// TIA Portal project "CPU1500_Profinet_PLC1_PLC2" (V16)

(* hardware
DEVICE "Station S71500/ET200MP_1"  S7-1500 station
   slot 0: "Châssis_0"  Rack  6ES7 590-1***0-0AA0
   slot 1: "PLC_1"  CPU 1511-1 PN  6ES7 511-1AK02-0AB0  V2.5
      slot 3: "Ecran CPU_1"  6ES7591-1AA00-0AA0
      slot 32768: "Interface PROFINET_1"  X1
         slot 32769: "Port_1"  X1 P1
         slot 32770: "Port_2"  X1 P2
   slot 2: "DI 32x24VDC BA_1"  DI 32x24VDC BA  6ES7 521-1BL10-0AA0  V1.0
   slot 3: "DQ 32x24VDC/0.5A BA_1"  DQ 32x24VDC/0.5A BA  6ES7 522-1BL10-0AA0  V1.0
DEVICE "Station S71500/ET200MP_2"  S7-1500 station
   slot 0: "Châssis_0"  Rack  6ES7 590-1***0-0AA0
   slot 1: "PLC_2"  CPU 1511-1 PN  6ES7 511-1AK01-0AB0  V2.1
      slot 3: "Ecran CPU_1"  6ES7591-1AA00-0AA0
      slot 32768: "Interface PROFINET_1"  X1
         slot 32769: "Port_1"  X1 P1
         slot 32770: "Port_2"  X1 P2
*)

// ===== PLC "PLC_1"  CPU 1511-1 PN =====

VAR_GLOBAL   // PLC tag table "Table de variables standard"
   "Clock_Byte" AT %MB0 : Byte;
   "Clock_10Hz" AT %M0.0 : Bool;
   "Clock_5Hz" AT %M0.1 : Bool;
   "Clock_2.5Hz" AT %M0.2 : Bool;
   "Clock_2Hz" AT %M0.3 : Bool;
   "Clock_1.25Hz" AT %M0.4 : Bool;
   "Clock_1Hz" AT %M0.5 : Bool;
   "Clock_0.625Hz" AT %M0.6 : Bool;
   "Clock_0.5Hz" AT %M0.7 : Bool;
END_VAR

DATA_BLOCK "DB_EMISSION"   // DB1
{ S7_Optimized_Access := 'FALSE' }
VERSION : 0.1
   VAR
      BOOL_0 : Bool;
      BOOL_1 : Bool;
      BOOL_2 : Bool;
      BOOL_3 : Bool;
      BOOL_4 : Bool;
      BOOL_5 : Bool;
      BOOL_6 : Bool;
      BOOL_7 : Bool;
      INT_0 : Int;
      INT_1 : Int;
      INT_2 : Int;
      INT_3 : Int;
      DINT_0 : DInt;
      DINT_1 : DInt;
      DINT_2 : DInt;
      DINT_3 : DInt;
   END_VAR
BEGIN
END_DATA_BLOCK

DATA_BLOCK "DB_RECEPTION"   // DB2
{ S7_Optimized_Access := 'FALSE' }
VERSION : 0.1
   VAR
      BOOL_0 : Bool;
      BOOL_1 : Bool;
      BOOL_2 : Bool;
      BOOL_3 : Bool;
      BOOL_4 : Bool;
      BOOL_5 : Bool;
      BOOL_6 : Bool;
      BOOL_7 : Bool;
      BOOL_8 : Bool;
      BOOL_9 : Bool;
      BOOL_10 : Bool;
      BOOL_11 : Bool;
      BOOL_12 : Bool;
      BOOL_13 : Bool;
      BOOL_14 : Bool;
      BOOL_15 : Bool;
      INT_0 : Int;
      INT_1 : Int;
      INT_2 : Int;
      INT_3 : Int;
      INT_4 : Int;
      INT_5 : Int;
      DINT_0 : DInt;
      DINT_1 : DInt;
      DINT_2 : DInt;
      DINT_3 : DInt;
      DINT_4 : DInt;
      DINT_5 : DInt;
      DINT_6 : DInt;
      DINT_7 : DInt;
      DINT_8 : DInt;
      DINT_9 : DInt;
      DINT_10 : DInt;
      DINT_11 : DInt;
   END_VAR
BEGIN
END_DATA_BLOCK

FUNCTION "FC_GEST_COM" : Void   // FC1, LAD
{ S7_Optimized_Access := 'TRUE' }
VERSION : 0.1
BEGIN

REGION Network 1
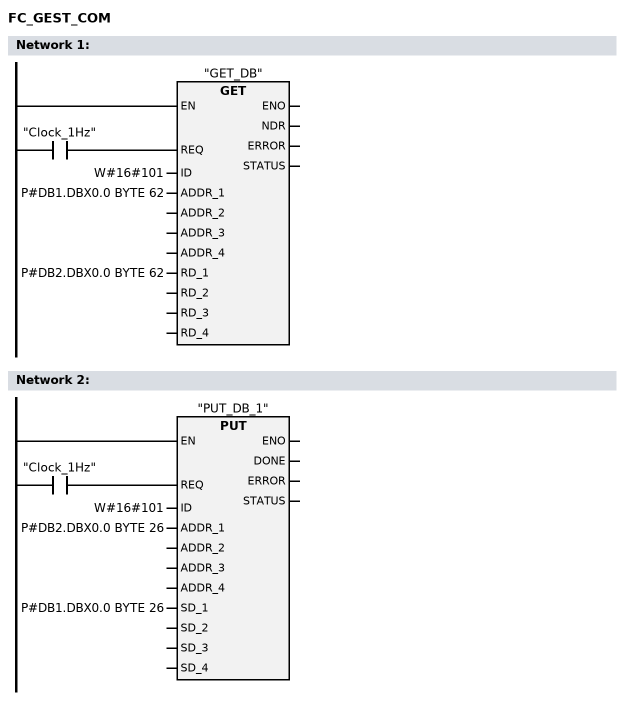
   "GET_DB"(REQ := "Clock_1Hz", ID := W#16#101, ADDR_1 := P#DB1.DBX0.0 BYTE 62, RD_1 := P#DB2.DBX0.0 BYTE 62);   // GET
END_REGION

REGION Network 2
   "PUT_DB_1"(REQ := "Clock_1Hz", ID := W#16#101, ADDR_1 := P#DB2.DBX0.0 BYTE 26, SD_1 := P#DB1.DBX0.0 BYTE 26);   // PUT
END_REGION
END_FUNCTION

ORGANIZATION_BLOCK "Main"   // OB1, LAD, ProgramCycle
TITLE = "Main Program Sweep (Cycle)"
{ S7_Optimized_Access := 'TRUE' }
VERSION : 0.1
   VAR_INPUT
      Initial_Call : Bool;   // Initial call of this OB
      Remanence : Bool;   // =True, if remanent data are available
   END_VAR
BEGIN

REGION Network 1: Appel du bloc FC de gestion de la communication
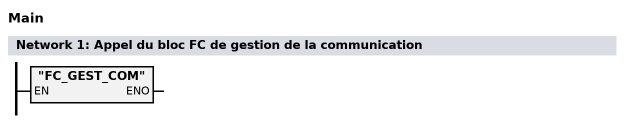
   RUNG wire#powerrail
      "FC_GEST_COM"()
   END_RUNG
   // the same network as SCL:
   "FC_GEST_COM"();
END_REGION
END_ORGANIZATION_BLOCK

// ===== PLC "PLC_2"  CPU 1511-1 PN =====

DATA_BLOCK "DB_EMISSION"   // DB1
{ S7_Optimized_Access := 'FALSE' }
VERSION : 0.1
   VAR
      BOOL_0 : Bool;
      BOOL_1 : Bool;
      BOOL_2 : Bool;
      BOOL_3 : Bool;
      BOOL_4 : Bool;
      BOOL_5 : Bool;
      BOOL_6 : Bool;
      BOOL_7 : Bool;
      BOOL_8 : Bool;
      BOOL_9 : Bool;
      BOOL_10 : Bool;
      BOOL_11 : Bool;
      BOOL_12 : Bool;
      BOOL_13 : Bool;
      BOOL_14 : Bool;
      BOOL_15 : Bool;
      INT_0 : Int;
      INT_1 : Int;
      INT_2 : Int;
      INT_3 : Int;
      INT_4 : Int;
      INT_5 : Int;
      DINT_0 : DInt;
      DINT_1 : DInt;
      DINT_2 : DInt;
      DINT_3 : DInt;
      DINT_4 : DInt;
      DINT_5 : DInt;
      DINT_6 : DInt;
      DINT_7 : DInt;
      DINT_8 : DInt;
      DINT_9 : DInt;
      DINT_10 : DInt;
      DINT_11 : DInt;
   END_VAR
BEGIN
END_DATA_BLOCK

DATA_BLOCK "DB_RECEPTION"   // DB2
{ S7_Optimized_Access := 'FALSE' }
VERSION : 0.1
   VAR
      BOOL_0 : Bool;
      BOOL_1 : Bool;
      BOOL_2 : Bool;
      BOOL_3 : Bool;
      BOOL_4 : Bool;
      BOOL_5 : Bool;
      BOOL_6 : Bool;
      BOOL_7 : Bool;
      INT_0 : Int;
      INT_1 : Int;
      INT_2 : Int;
      INT_3 : Int;
      DINT_0 : DInt;
      DINT_1 : DInt;
      DINT_2 : DInt;
      DINT_3 : DInt;
   END_VAR
BEGIN
END_DATA_BLOCK

ORGANIZATION_BLOCK "Main"   // OB1, LAD, ProgramCycle
TITLE = "Main Program Sweep (Cycle)"
{ S7_Optimized_Access := 'TRUE' }
VERSION : 0.1
   VAR_INPUT
      Initial_Call : Bool;   // Initial call of this OB
      Remanence : Bool;   // =True, if remanent data are available
   END_VAR
BEGIN
END_ORGANIZATION_BLOCK